(* IEC 61131-3 sources: Industry-PLC-LLM/data/PLCBEAD_repo/PLCBEAD_PLCEmbed-main/PLC-BEAD/Source/GEB/building_PULSE_LENGTH, 1 file *)

(* ---- PULSE_LENGTH.ST ---- *)
FUNCTION UDINT_TO_TIME2:TIME

	VAR_INPUT
		IN :	UDINT;
	END_VAR

	UDINT_TO_TIME2 := DINT_TO_TIME(UDINT_TO_DINT(IN));

END_FUNCTION

FUNCTION_BLOCK T_PLC_MS_block
	VAR_OUTPUT
		T_PLC_MS :	UDINT;
	END_VAR

	VAR
		PLC_TICKS_PER_SEC :	INT;
		PLC_SYS_TICK_CNT :	DINT;
	END_VAR

	VAR
		debug :	BOOL;(*Debug-Mode ON / OFF*)
		N :	INT;(*Debug-Faktor*)
		Offset :	UDINT;(*Debug-Offset*)
		temp :	DWORD := DWORD#1;(*Debug-Offset*)
		MODE :	BOOL;(*modus*)
		faktor :	UDINT;(*Systemtakt-Faktor*)
		init :	BOOL;
		v_plc_ticks_per_sec :	UDINT;
		base :	UDINT := UDINT#1000;
	END_VAR

	IF init = FALSE THEN
		v_plc_ticks_per_sec := INT_TO_UDINT(PLC_TICKS_PER_SEC);
		IF v_plc_ticks_per_sec = UDINT#1024 THEN
			faktor := UDINT#1;
			MODE := FALSE;
		ELSIF v_plc_ticks_per_sec > UDINT#0 THEN
			IF v_plc_ticks_per_sec <= base THEN
				faktor := base / v_plc_ticks_per_sec;
				MODE := FALSE;
			ELSE
				faktor := v_plc_ticks_per_sec / base;
				MODE := TRUE;
			END_IF;
		ELSE
			faktor := UDINT#1;
		END_IF;
		init := TRUE;
	END_IF;

	IF MODE THEN
		T_PLC_MS := DINT_TO_UDINT(PLC_SYS_TICK_CNT) / faktor;
	ELSE
		T_PLC_MS := DINT_TO_UDINT(PLC_SYS_TICK_CNT) * faktor;
	END_IF;

	IF debug THEN
		T_PLC_MS := (DWORD_TO_UDINT(SHL(UDINT_TO_DWORD(T_PLC_MS),N) OR SHL(temp,N)) - UDINT#1) + Offset;
	END_IF;

END_FUNCTION_BLOCK

FUNCTION_BLOCK PULSE_LENGTH_Block

	VAR_INPUT
		IN :	BOOL;
		T_SHORT :	TIME := T#100ms;
		T_LONG :	TIME := T#1s;
	END_VAR

	VAR_OUTPUT
		SHORT :	BOOL;
		MIDDLE :	BOOL;
		LONG :	BOOL;
	END_VAR

	VAR
		TX :	TIME;
		tn :	TIME;
		edge :	BOOL;
		T_PLC_MS :	T_PLC_MS_block;
	END_VAR

	T_PLC_MS();
	TX:= UDINT_TO_TIME(T_PLC_MS.T_PLC_MS);

	short := FALSE;
	MidDLe := FALSE;
	long := FALSE;

	IF IN AND NOT edge THEN
		edge := TRUE;
		tn := TX;

	ELSIF NOT IN AND edge THEN
		edge := FALSE;
		tn := TX - tn;
		IF tn < t_short THEN
			short := TRUE;
		ELSIF tn > t_long THEN
			long := TRUE;
		ELSE
			MidDLe := TRUE;
		END_IF;

	ELSIF IN AND TX - tn > t_long THEN
		long := TRUE;
	END_IF;

END_FUNCTION_BLOCK

PROGRAM program0
	VAR
		IN :	BOOL;
		T_SHORT :	TIME := T#100ms;
		T_LONG :	TIME := T#1s;
		SHORT :	BOOL;
		MIDDLE :	BOOL;
		LONG :	BOOL;

		func_block : PULSE_LENGTH_Block;
	END_VAR
	func_block.IN := IN;
	func_block.T_SHORT := T_SHORT;
	func_block.T_LONG := T_LONG ;

	func_block();
	SHORT  := func_block.SHORT;
	MIDDLE  := func_block.MIDDLE;
	LONG  := func_block.LONG;
END_PROGRAM
